(*
SPDX-FileCopyrightText: © 2026 Oleksandr Tiutyk <trofimich@gmail.com>
SPDX-License-Identifier: MIT
License: https://opensource.org/license/mit
*)

(*!
<summary>Provides workflow node creation, transition validation, topology checks and configuration helpers.</summary>
<description>
Public facade delegating element creation and type description to WorkflowElementFactory, state-transition and
attachment validation to WorkflowElementHelper, and configuration serialization helpers to
WorkflowConfigurationSerializer.
Defines the canonical transition table for WORKFLOW_ELEMENT_STATE. Fresh starts require PASSIVE_READY,
resuming requires PASSIVE_SUSPENDED, and completed, halted, cancelled or failed elements must pass through
ACTIVE_RESETTING before returning to PASSIVE_READY.
</description>
*)

{attribute 'no_explicit_call' := 'do not call this function block directly'}
PROGRAM Workflows
VAR CONSTANT
	//! <summary>No activity or branch is selected; never pass this value to a nonnegative index input.</summary>
	//! <description>
	//! SequenceActivity and WaitAndPickActivity expose this DINT sentinel while selection is absent.
	//! </description>
	NO_SELECTED_ACTIVITY_INDEX : DINT := -1;
END_VAR
VAR
	{attribute 'hide'} 
	_ClassName : STRING := __POUNAME();
END_VAR

(*!
<summary>Returns the program name for diagnostic reporting.</summary>
*)
{attribute 'monitoring' := 'call'}
PROPERTY ClassName : REFERENCE TO STRING
GET
ClassName REF= _ClassName;
END_GET
END_PROPERTY

(*!
<summary>Returns the elementary IEC spelling used in configuration documents.</summary>
<description>String capacities exclude the terminator. Unsupported types raise before writing the value.</description>
*)
METHOD ConfigurationTypeName : STRING
VAR_INPUT
	typeClass : __SYSTEM.TYPE_CLASS;
	size : UDINT;
END_VAR
ConfigurationTypeName := WorkflowElementFactory.ConfigurationTypeName(
	typeClass := typeClass,
	size := size
);
END_METHOD

(*!
<summary>Maps an elementary IEC type class to its CONFIGURATION_VALUE_TYPE enum.</summary>
<description>Unsupported type classes raise a configuration exception.</description>
<param name="typeClass">Type class from __SYSTEM.TYPE_CLASS.</param>
*)
METHOD ConfigurationValueType : TOF_Core.CONFIGURATION_VALUE_TYPE
VAR_INPUT
	typeClass : __SYSTEM.TYPE_CLASS;
END_VAR
ConfigurationValueType := WorkflowElementFactory.ConfigurationValueType(
	typeClass := typeClass
);
END_METHOD

(*!
<summary>Creates a dynamic workflow element and returns it after ownership registration.</summary>
<description>Requires a live ready workflow in its owning task. Built-in qualified names are handled first, then the
optional application factory. Unknown names raise a configuration exception. A successful element is borrowed
until workflow disposal; configuration and attachment are separate operations. Registration failures propagate
under the RegisterChild cleanup contract. Call outside lifecycle methods and without reentry.</description>
<param name="typeName">Case-sensitive qualified PLC type.</param>
<param name="workflow">Owner of the resulting element.</param>
<param name="factory">Optional application type factory.</param>
*)
METHOD CreateElement : IWorkflowElement
VAR_INPUT
	typeName : STRING(255);
	workflow : IWorkflow;
	factory : IWorkflowElementFactory := 0;
END_VAR
CreateElement := WorkflowElementFactory.CreateElement(
	typeName := typeName,
	workflow := workflow,
	factory := factory
);
END_METHOD

(*!
<summary>Borrows an IEC variable as a typed initial element descriptor.</summary>
<description>Keep the source alive and unchanged through DeclareArray. The descriptor carries the exact IEC category
and full storage width. No allocation or ownership transfer occurs.</description>
<param name="value">Live typed PLC variable.</param>
*)
METHOD GetValueDescriptor : __SYSTEM.AnyType
VAR_INPUT
	value : ANY;
END_VAR
GetValueDescriptor := value;
END_METHOD

(*!
<summary>Resolves an exact elementary type and storage capacity.</summary>
<description>Use within one synchronous load. Handles borrow the active document and expire when it is replaced.</description>
*)
METHOD ParseTypeDescriptor : __SYSTEM.AnyType
VAR_INPUT
	typeName : STRING;
END_VAR
ParseTypeDescriptor := WorkflowElementFactory.ParseTypeDescriptor(typeName := typeName);
END_METHOD

(*!
<summary>Returns a comma-separated list of target states permitted from the given state.</summary>
<description>
Lists targets accepted by ValidateTransition in diagnostic display order.
</description>
<param name="currentState">Current state of the workflow element.</param>
*)
METHOD GetAllowedTransitionNames : STRING(255)
VAR_INPUT
	currentState : WORKFLOW_ELEMENT_STATE;
END_VAR
GetAllowedTransitionNames := WorkflowElementHelper.GetAllowedTransitionNames(
	currentState := currentState
);
END_METHOD

(*!
<summary>Returns the library namespace name for diagnostic reporting.</summary>
*)
{attribute 'monitoring' := 'call'}
PROPERTY NamespaceName : REFERENCE TO STRING
GET
NamespaceName REF= CurrentNamespace.Name;
END_GET
END_PROPERTY

(*!
<summary>Restores a child and checks the interface required by its parent role.</summary>
<description>Use within one synchronous load. Handles borrow the active document and expire when it is replaced.</description>
<param name="loader">Workflow loader providing element construction services.</param>
<param name="node">Configuration node of the activity.</param>
*)
METHOD ReadActivity : IActivity
VAR_INPUT
	loader : IWorkflowLoader;
	node : TOF_Core.CONFIGURATION_NODE;
END_VAR
ReadActivity := WorkflowConfigurationSerializer.ReadActivity(
	loader := loader,
	node := node
);
END_METHOD

(*!
<summary>Restores a child and checks the interface required by its parent role.</summary>
<description>Use within one synchronous load. Handles borrow the active document and expire when it is replaced.</description>
<param name="loader">Workflow loader providing element construction services.</param>
<param name="node">Configuration node of the catch activity.</param>
*)
METHOD ReadCatchActivity : ICatchActivity
VAR_INPUT
	loader : IWorkflowLoader;
	node : TOF_Core.CONFIGURATION_NODE;
END_VAR
ReadCatchActivity := WorkflowConfigurationSerializer.ReadCatchActivity(
	loader := loader,
	node := node
);
END_METHOD

(*!
<summary>Restores a child and checks the interface required by its parent role.</summary>
<description>Use within one synchronous load. Handles borrow the active document and expire when it is replaced.</description>
<param name="loader">Workflow loader providing element construction services.</param>
<param name="node">Configuration node of the condition.</param>
*)
METHOD ReadCondition : ICondition
VAR_INPUT
	loader : IWorkflowLoader;
	node : TOF_Core.CONFIGURATION_NODE;
END_VAR
ReadCondition := WorkflowConfigurationSerializer.ReadCondition(
	loader := loader,
	node := node
);
END_METHOD

(*!
<summary>Reads local variable declarations and the display name for a named workflow object.</summary>
<description>Restores local declarations into scope and reads the 'name' field into target.Name.
Use within one synchronous load.</description>
<param name="reader">Active configuration reader.</param>
<param name="node">Configuration object node.</param>
<param name="target">Named workflow object receiving the restored display name.</param>
<param name="scope">Declaration container receiving local variable declarations.</param>
*)
METHOD ReadConfigurationHeader
VAR_INPUT
	reader : TOF_Core.IConfigurationReader;
	node : TOF_Core.CONFIGURATION_NODE;
	target : TOF_Core.INamed;
	scope : IDeclaredVariableContainer;
END_VAR
WorkflowConfigurationSerializer.ReadConfigurationHeader(
	reader := reader,
	node := node,
	target := target,
	scope := scope
);
END_METHOD

(*!
<summary>Copies all initial declarations into a fresh local scope.</summary>
<description>Use within one synchronous load. Handles borrow the active document and expire when it is replaced.</description>
<param name="reader">Active configuration reader.</param>
<param name="node">Configuration object node.</param>
<param name="scope">Declaration container receiving local variable declarations.</param>
*)
METHOD ReadDeclarations
VAR_INPUT
	reader : TOF_Core.IConfigurationReader;
	node : TOF_Core.CONFIGURATION_NODE;
	scope : IDeclaredVariableContainer;
END_VAR
WorkflowConfigurationSerializer.ReadDeclarations(
	reader := reader,
	node := node,
	scope := scope
);
END_METHOD

(*!
<summary>Allocates and decodes a literal into caller-owned byte storage.</summary>
<description>Use within one synchronous load. Handles borrow the active document and expire when it is replaced.</description>
<param name="reader">Active configuration reader.</param>
<param name="node">Configuration node containing literal object.</param>
*)
METHOD ReadLiteral : __SYSTEM.AnyType
VAR_INPUT
	reader : TOF_Core.IConfigurationReader;
	node : TOF_Core.CONFIGURATION_NODE;
END_VAR
ReadLiteral := WorkflowConfigurationSerializer.ReadLiteral(
	reader := reader,
	node := node
);
END_METHOD

(*!
<summary>Reads an IEC name without truncation.</summary>
<description>The reader rejects an oversized field.</description>
<param name="reader">Active configuration reader.</param>
<param name="node">Configuration node containing string name.</param>
*)
METHOD ReadName : STRING
VAR_INPUT
	reader : TOF_Core.IConfigurationReader;
	node : TOF_Core.CONFIGURATION_NODE;
END_VAR
ReadName := WorkflowConfigurationSerializer.ReadName(
	reader := reader,
	node := node
);
END_METHOD

(*!
<summary>Reads a qualified configuration type name.</summary>
<description>Use within one synchronous load. Handles borrow the active document and expire when it is replaced.</description>
<param name="reader">Active configuration reader.</param>
<param name="node">Configuration node containing type name.</param>
*)
METHOD ReadTypeName : STRING(255)
VAR_INPUT
	reader : TOF_Core.IConfigurationReader;
	node : TOF_Core.CONFIGURATION_NODE;
END_VAR
ReadTypeName := WorkflowConfigurationSerializer.ReadTypeName(
	reader := reader,
	node := node
);
END_METHOD

(*!
<summary>Restores a child and checks the interface required by its parent role.</summary>
<description>Use within one synchronous load. Handles borrow the active document and expire when it is replaced.</description>
<param name="loader">Workflow loader providing element construction services.</param>
<param name="node">Configuration node of the condition.</param>
*)
METHOD ReadVariableHasValueCondition : IVariableHasValueCondition
VAR_INPUT
	loader : IWorkflowLoader;
	node : TOF_Core.CONFIGURATION_NODE;
END_VAR
ReadVariableHasValueCondition := WorkflowConfigurationSerializer.ReadVariableHasValueCondition(
	loader := loader,
	node := node
);
END_METHOD

(*!
<summary>Validates a borrowed parent-child link before any graph mutation.</summary>
<description>
Rejects nulls, self or ancestor cycles, a different existing parent, non-ready activity ancestors or children,
and a non-ready owning workflow. A child with a known workflow requires a parent with that same known owner;
an unassociated subtree may inherit its owner after attachment. This prevents hiding associated descendants
inside an unassociated subtree. Configure may reuse a link to this parent; append APIs separately reject any
occupied child slot. Does not detach, transfer ownership or mutate either operand. Caller callbacks and
metadata must obey their single-task, no-reentry and lifetime contracts.
</description>
<param name="parent">Live prospective parent.</param>
<param name="child">Live child candidate whose link is being validated.</param>
*)
METHOD INTERNAL ValidateElementAttachment
VAR_INPUT
	parent : IWorkflowElement;
	child : IWorkflowElement;
END_VAR
WorkflowElementHelper.ValidateElementAttachment(
	parent := parent,
	child := child
);
END_METHOD

(*!
<summary>Reports whether transitioning from currentState to newState is permitted.</summary>
<description>
Does not mutate state or raise exceptions. Callers use this predicate before changing state or validating
external requests.
</description>
<param name="currentState">Current state of the workflow element.</param>
<param name="newState">Requested target state.</param>
*)
METHOD ValidateTransition : BOOL
VAR_INPUT
	currentState : WORKFLOW_ELEMENT_STATE;
	newState : WORKFLOW_ELEMENT_STATE;
END_VAR
ValidateTransition := WorkflowElementHelper.ValidateTransition(
	currentState := currentState,
	newState := newState
);
END_METHOD

(*!
<summary>Writes qualified type, display name and local declarations for one node.</summary>
<description>Call once per node before writing its configuration fields. Only owned declarations are enumerated.</description>
*)
METHOD WriteConfigurationHeader
VAR_INPUT
	writer : TOF_Core.IConfigurationWriter;
	source : TOF_Core.IObject;
	displayName : WSTRING;
	scope : IDeclaredVariableContainer;
END_VAR
WorkflowConfigurationSerializer.WriteConfigurationHeader(
	writer := writer,
	source := source,
	displayName := displayName,
	scope := scope
);
END_METHOD

(*!
<summary>Writes the type and value of a configured literal operand.</summary>
<description>The source descriptor is borrowed for this call. Unsupported types raise.</description>
*)
METHOD WriteConfigurationLiteral
VAR_INPUT
	writer : TOF_Core.IConfigurationWriter;
	name : STRING;
	value : __SYSTEM.AnyType;
END_VAR
WorkflowConfigurationSerializer.WriteConfigurationLiteral(
	writer := writer,
	name := name,
	value := value
);
END_METHOD

(*!
<summary>Writes a nested configuration under the supplied role.</summary>
<description>
The object must implement the serialization interface. Null mandatory objects and unsupported objects raise.
</description>
*)
METHOD WriteConfigurationObject
VAR_INPUT
	writer : TOF_Core.IConfigurationWriter;
	name : STRING;
	source : TOF_Core.IObject;
END_VAR
WorkflowConfigurationSerializer.WriteConfigurationObject(
	writer := writer,
	name := name,
	source := source
);
END_METHOD

(*!
<summary>Writes one embedded configuration or one stable external key.</summary>
<description>
An unspecified binding raises with the node name. Borrowed objects need no serialization interface.
</description>
*)
METHOD WriteDependency
VAR_INPUT
	writer : TOF_Core.IConfigurationWriter;
	role : STRING;
	kind : DEPENDENCY_BINDING_KIND;
	key : STRING;
	dependency : TOF_Core.IObject;
	nodeName : WSTRING;
END_VAR
WorkflowConfigurationSerializer.WriteDependency(
	writer := writer,
	role := role,
	kind := kind,
	key := key,
	dependency := dependency,
	nodeName := nodeName
);
END_METHOD

(*!
<summary>Formats a comparison operator enumeration value into its standard string representation.</summary>
<description>Delegates to WorkflowConfigurationSerializer.</description>
<param name="comparisonOperator">Comparison operator to format.</param>
*)
METHOD FormatComparisonOperator : STRING
VAR_INPUT
	comparisonOperator : COMPARISON_OPERATOR;
END_VAR
FormatComparisonOperator := WorkflowConfigurationSerializer.FormatComparisonOperator(
	comparisonOperator := comparisonOperator
);
END_METHOD

(*!
<summary>Formats a logical operator enumeration value into its standard uppercase string representation.</summary>
<description>Delegates to WorkflowConfigurationSerializer.</description>
<param name="logicalOperator">Logical operator to format.</param>
*)
METHOD FormatLogicalOperator : STRING
VAR_INPUT
	logicalOperator : LOGICAL_OPERATOR;
END_VAR
FormatLogicalOperator := WorkflowConfigurationSerializer.FormatLogicalOperator(
	logicalOperator := logicalOperator
);
END_METHOD

(*!
<summary>Parses a comparison operator from its string representation.</summary>
<description>Delegates to WorkflowConfigurationSerializer.</description>
<param name="rawOperator">Operator string to parse.</param>
*)
METHOD ParseComparisonOperator : COMPARISON_OPERATOR
VAR_INPUT
	rawOperator : STRING;
END_VAR
ParseComparisonOperator := WorkflowConfigurationSerializer.ParseComparisonOperator(
	rawOperator := rawOperator
);
END_METHOD

(*!
<summary>Parses a logical operator from its string representation.</summary>
<description>Delegates to WorkflowConfigurationSerializer.</description>
<param name="rawOperator">Operator string to parse.</param>
*)
METHOD ParseLogicalOperator : LOGICAL_OPERATOR
VAR_INPUT
	rawOperator : STRING;
END_VAR
ParseLogicalOperator := WorkflowConfigurationSerializer.ParseLogicalOperator(
	rawOperator := rawOperator
);
END_METHOD

END_PROGRAM

(* stored: Version 1.1.0.1
   POU Workflows: Id {09179207-e85a-4ce9-a60e-213a99d7b743}, SpecialFunc None
   Folder Service methods: Id {84931a7b-3d4a-4632-9cb1-e5d7a8f192b4}
   Property ClassName: Id {481cf308-45d8-4e8a-9beb-4d74c6f3cadc}
   Get Get: Id {d4104013-1803-475d-a0e1-512983ee4a03}
   Method ConfigurationTypeName: Id {e19b9cf7-a009-4705-aacb-39f7d6d97cc6}
   Method ConfigurationValueType: Id {b888840e-ea36-4c5a-b4fa-e0d8dd9a7b2a}
   Method CreateElement: Id {693894bc-56da-47d7-b359-9e37c1dedefe}
   Method GetValueDescriptor: Id {4fae6f9f-c8bd-454e-aa6a-dfa4443d6513}
   Method ParseTypeDescriptor: Id {bed09c9b-1f24-4dbb-9ac1-8c3c77270d19}
   Method GetAllowedTransitionNames: Id {41bf9062-9c5f-4633-8ce3-cbe75b618334}
   Property NamespaceName: Id {f189a98d-babc-4b35-b814-9f960e872687}
   Get Get: Id {7cc74d8e-6055-476f-8cf2-6211037db96f}
   Method ReadActivity: Id {98f68397-5f00-4cef-a8c2-0506c6c4e202}
   Method ReadCatchActivity: Id {8c543632-4522-4db9-9268-45235c983784}
   Method ReadCondition: Id {775db239-85c0-4318-a235-4deda689de89}
   Method ReadConfigurationHeader: Id {c18d4e92-3a7b-4f60-85c1-92d4e6b8a0f3}
   Method ReadDeclarations: Id {869b056d-ad87-4e0a-9f82-e70f970b435e}
   Method ReadLiteral: Id {30a44b32-53cb-4c18-ad77-87a97061ecc3}
   Method ReadName: Id {88e9b459-6768-4c73-8437-11b767b5356c}
   Method ReadTypeName: Id {35ac909b-9386-4cf0-8aee-a7908186761d}
   Method ReadVariableHasValueCondition: Id {ab79eafb-a2eb-4395-8ac6-d5069fde64a9}
   Method ValidateElementAttachment: Id {39a48f34-ab25-4bc8-a7ce-16ed935b5b85}
   Method ValidateTransition: Id {bc368e59-28e8-40f0-ada3-0cec58c2ed3a}
   Method WriteConfigurationHeader: Id {636274aa-4460-45bb-b93e-ab61e0c5c633}
   Method WriteConfigurationLiteral: Id {6e4854ec-3314-41e0-a392-502ce654358b}
   Method WriteConfigurationObject: Id {b5a855d9-a98e-4518-b7a1-32b28d730a95}
   Method WriteDependency: Id {ba1e2d68-647b-4258-ba55-41eaae9d44b5}
   Method FormatComparisonOperator: Id {fbf344a9-0aff-4f5e-a0fa-5a4effb181ba}
   Method FormatLogicalOperator: Id {d82116e3-9bff-4d4b-89a0-3db4c0f573ea}
   Method ParseComparisonOperator: Id {5c24df7e-997b-4182-9ed0-a17b299b3d91}
   Method ParseLogicalOperator: Id {b0bb9f0f-3d04-4a21-8523-6bb1ca1bbbbe} *)
